// TIA Portal V17 export
// export: Created 2023-09-11T20:22:11.5433454Z, ExportSetting WithDefaults, DisplayName Totally Integrated Automation Portal, DisplayVersion V17 Update 6, DisplayName TIA Portal Openness, DisplayVersion V17 Update 6, DisplayName TIA Portal Teamcenter Gateway, DisplayVersion V17 Update 6, DisplayName TIA Portal Version Control Interface, DisplayVersion V17, DisplayName Simotion SCOUT TIA, DisplayVersion 5.4.3.0, DisplayName TIA Portal Test Suite Advanced, DisplayVersion V17 Update 1, DisplayName SIMOCODE ES, DisplayVersion V17 Update 5, DisplayName SINAMICS Startdrive Advanced, DisplayVersion V17 SP1, DisplayName SINAMICS Startdrive G130, G150, S120, S150, SINAMICS MV, S210, DisplayVersion V17 SP1, DisplayName SINAMICS Startdrive G110M, G120, G120C, G120D, G120P, G115D, DisplayVersion V17 SP1, DisplayName SIRIUS Safety ES, DisplayVersion V17 Update 5, DisplayName STEP 7 Professional, DisplayVersion V17 Update 6, DisplayName STEP 7 CFC, DisplayVersion V17 Update 1, DisplayName STEP 7 Safety, DisplayVersion V17 Update 6, DisplayName WinCC Advanced, DisplayVersion V17 Update 6, DisplayName SIMATIC Visualization Architect, DisplayVersion V17 Update 5
FUNCTION "07_Speed Control" : Void   // FC8, F_LAD
TITLE = Manage Safety Encoder
{ S7_Optimized_Access := 'TRUE' }
VERSION : 0.1
// stored: AutoNumber true, IsIECCheckEnabled false, UDAEnableTagReadback false
BEGIN

REGION Network 1: !!COLUMN_1$$
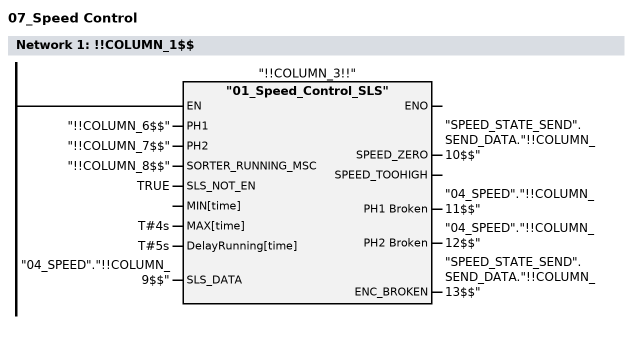
   RUNG wire#powerrail
      "!!COLUMN_3!!"(PH1 := "!!COLUMN_6$$", PH2 := "!!COLUMN_7$$", SORTER_RUNNING_MSC := "!!COLUMN_8$$", SLS_NOT_EN := TRUE, "MIN[time]" :=, "MAX[time]" := T#4s, "DelayRunning[time]" := T#5s, SLS_DATA := "04_SPEED"."!!COLUMN_9$$", SPEED_ZERO => "SPEED_STATE_SEND".SEND_DATA."!!COLUMN_10$$", SPEED_TOOHIGH =>, "PH1 Broken" => "04_SPEED"."!!COLUMN_11$$", "PH2 Broken" => "04_SPEED"."!!COLUMN_12$$", ENC_BROKEN => "SPEED_STATE_SEND".SEND_DATA."!!COLUMN_13$$")
   END_RUNG
   // the same network as SCL:
   "!!COLUMN_3!!"(PH1 := "!!COLUMN_6$$",   // "01_Speed_Control_SLS"
                  PH2 := "!!COLUMN_7$$",
                  SORTER_RUNNING_MSC := "!!COLUMN_8$$",
                  SLS_NOT_EN := TRUE,
                  "MAX[time]" := T#4s,
                  "DelayRunning[time]" := T#5s,
                  SLS_DATA := "04_SPEED"."!!COLUMN_9$$",
                  SPEED_ZERO => "SPEED_STATE_SEND".SEND_DATA."!!COLUMN_10$$",
                  "PH1 Broken" => "04_SPEED"."!!COLUMN_11$$",
                  "PH2 Broken" => "04_SPEED"."!!COLUMN_12$$",
                  ENC_BROKEN => "SPEED_STATE_SEND".SEND_DATA."!!COLUMN_13$$");
END_REGION
END_FUNCTION
